// TwinCAT 3 PLC project PLCProject
// ProgramVersion: 3.1.4024.0
// libraries:
//   Tc2_MC2, * (Beckhoff Automation GmbH)
//   Tc2_NCI, * (Beckhoff Automation GmbH)
//   Tc2_NcKinematicTransformation, * (Beckhoff Automation GmbH)
//   Tc2_Standard, * (Beckhoff Automation GmbH)
//   Tc2_System, * (Beckhoff Automation GmbH)
//   Tc3_Module, * (Beckhoff Automation GmbH)
// project tree:
//   DUTs/ UI_TO_PLC.TcDUT, PLC_TO_UI.TcDUT
//   GVLs/ UIData.TcGVL
//   / PlcTask.TcTTO
//   POUs/FunctionBlock/ FB_EnableAxes.TcPOU, FB_LoadFileRun.TcPOU, FB_MachineCodeHandling.TcPOU, FB_NCIChannelGrouping.TcPOU, LifeBitMonitor.TcPOU
//   POUs/ MAIN.TcPOU
//   POUs/Programs/ Delta_Robot_Program.TcPOU
// real-time tasks:
//   TASK PlcTask: cycle T#10ms, priority 20, ADS port 350
// motion (NC):
//   TASK NC-Task 1 SAF: cycle T#2ms, priority 4, ADS port 501
//   TASK NC-Task 1 SVB: cycle T#10ms, priority 8, ADS port 511
//   AXIS X_MCS (id 1)
//   AXIS Y_MCS (id 2)
//   AXIS Z_MCS (id 3)
//   AXIS M1_ACS (id 4)
//     OtherSettings: AllowMotionCmdToSlave=true
//     encoder EncType=1
//     drive DrvType=5
//       Analog: TorqueSetpointScale=10, ScaleFactorActTorque=0.1
//     controller CtrType=1
//       CtrPara: PriorControlFactor=1
//         Observer: BandWidth=20
//   AXIS M2_ACS (id 5)
//     OtherSettings: AllowMotionCmdToSlave=true
//     encoder EncType=1
//     drive DrvType=5
//       Analog: TorqueSetpointScale=10, ScaleFactorActTorque=0.1
//     controller CtrType=1
//       CtrPara: PriorControlFactor=1
//         Observer: BandWidth=20
//   AXIS M3_ACS (id 6)
//     OtherSettings: AllowMotionCmdToSlave=true
//     encoder EncType=1
//     drive DrvType=5
//       Analog: TorqueSetpointScale=10, ScaleFactorActTorque=0.1
//     controller CtrType=1
//       CtrPara: PriorControlFactor=1
//         Observer: BandWidth=20
// variable links:
//   PLCProject Instance <-> NC-Task 1 SAF/Axes/M1_ACS
//     PlcTask Inputs/Delta_Robot_Program.io_M1.NcToPlc <-> Outputs/ToPlc
//     PlcTask Outputs/Delta_Robot_Program.io_M1.PlcToNc <-> Inputs/FromPlc
//   PLCProject Instance <-> NC-Task 1 SAF/Axes/M2_ACS
//     PlcTask Inputs/Delta_Robot_Program.io_M2.NcToPlc <-> Outputs/ToPlc
//     PlcTask Outputs/Delta_Robot_Program.io_M2.PlcToNc <-> Inputs/FromPlc
//   PLCProject Instance <-> NC-Task 1 SAF/Axes/M3_ACS
//     PlcTask Inputs/Delta_Robot_Program.io_M3.NcToPlc <-> Outputs/ToPlc
//     PlcTask Outputs/Delta_Robot_Program.io_M3.PlcToNc <-> Inputs/FromPlc
//   PLCProject Instance <-> NC-Task 1 SAF/Axes/X_MCS
//     PlcTask Inputs/Delta_Robot_Program.io_X.NcToPlc <-> Outputs/ToPlc
//     PlcTask Outputs/Delta_Robot_Program.io_X.PlcToNc <-> Inputs/FromPlc
//   PLCProject Instance <-> NC-Task 1 SAF/Axes/Y_MCS
//     PlcTask Inputs/Delta_Robot_Program.io_Y.NcToPlc <-> Outputs/ToPlc
//     PlcTask Outputs/Delta_Robot_Program.io_Y.PlcToNc <-> Inputs/FromPlc
//   PLCProject Instance <-> NC-Task 1 SAF/Axes/Z_MCS
//     PlcTask Inputs/Delta_Robot_Program.io_Z.NcToPlc <-> Outputs/ToPlc
//     PlcTask Outputs/Delta_Robot_Program.io_Z.PlcToNc <-> Inputs/FromPlc
//   PLCProject Instance <-> NC-Task 1 SAF/KinematicChannel
//     PlcTask Inputs/Delta_Robot_Program.in_stKinToPlc <-> Outputs/ToPlc
//     PlcTask Outputs/Delta_Robot_Program.out_stPlcToKin <-> Inputs/FromPlc
//   PLCProject Instance <-> NC-Task 1 SAF/NCIChannel
//     PlcTask Inputs/Delta_Robot_Program.in_stItpToPlc <-> Outputs/ToPlc
//     PlcTask Outputs/Delta_Robot_Program.out_stPlcToItp <-> Inputs/FromPlc

CONFIGURATION PLCProject
    RESOURCE PLC ON TwinCAT3
        TASK PlcTask(INTERVAL := T#10ms, PRIORITY := 20);
        PROGRAM MAIN WITH PlcTask : MAIN;
    END_RESOURCE
END_CONFIGURATION

// ---- DUTs/UI_TO_PLC.TcDUT
TYPE UI_TO_PLC :
STRUCT
	EnableMonitoring : BOOL;
	LifeBit : BOOL;
	EnableAllAxis : BOOL;
	ResetAllAxis : BOOL;
	ConfigKinematicGroup :BOOL;
	ResetKinematicGroup : BOOL;
	XJogPositive : BOOL;
	YJogPositive : BOOL;
	ZJogPositive : BOOL;
	XJogNegative : BOOL;
	YJogNegative : BOOL;
	ZJogNegative : BOOL;
	JogSpeed     : REAL;
	NCIAxisGroup : BOOL;
	NCIAxisUnGroup : BOOL;
	NCIInteperatorReset : BOOL;
	RunPartProgram : BOOL;
	StopPartProgram : BOOL;
	NCIOverRidePer : REAL;
	PartProgramName : STRING(80);
END_STRUCT
END_TYPE

// ---- DUTs/PLC_TO_UI.TcDUT
TYPE PLC_TO_UI :
STRUCT
	X_MCSPos : REAL;
	Y_MCSPos : REAL;
	Z_MCSPos : REAL;
	M1_ACSPos : REAL;
	M2_ACSPos : REAL;
	M3_ACSPos : REAL;
	AllAxisEnabled : BOOL;
	AxisError : BOOL;
	KinematicGroupError : BOOL;	
	KinematicGroupingReady : BOOL;
	NCIAxisGrouped : BOOL;
	NCIAXisError : BOOL;
	NCIInterpreterState : UDINT;
	PartProgramLine1 : STRING(80);
	PartProgramLine2 : STRING(80);
	PartProgramLine3 : STRING(80);
END_STRUCT
END_TYPE

// ---- GVLs/UIData.TcGVL
{attribute 'qualified_only'}
VAR_GLOBAL
	stUI_TO_PLC : UI_TO_PLC;
	stPLC_TO_UI : PLC_TO_UI;
END_VAR

// ---- POUs/MAIN.TcPOU
PROGRAM MAIN
VAR
END_VAR

Delta_Robot_Program();

END_PROGRAM

// ---- POUs/Programs/Delta_Robot_Program.TcPOU
PROGRAM Delta_Robot_Program
VAR	
	(* Axis Enable *)
	fbEnableAxes				: FB_EnableAxes;
	io_X						: AXIS_REF;
	io_Y						: AXIS_REF;
	io_Z						: AXIS_REF;
	io_M1						: AXIS_REF;
	io_M2						: AXIS_REF;
	io_M3						: AXIS_REF;
	bEnableAxes: BOOL;
	bAllAxesReady: BOOL;
	bAxisError: BOOL;
	bResetAxes: BOOL;
	
	(* Kinematics *)
	in_stKinToPlc	AT %I*		: NCTOPLC_NCICHANNEL_REF;
	out_stPlcToKin	AT %Q*		: PLCTONC_NCICHANNEL_REF;
	fbConfigKinGroup      		: FB_KinConfigGroup;
    stAxesConfig          		: ST_KinAxes;
	fbResetKinGroup				: FB_KinResetGroup;
	bConfigKinematicGroup: BOOL;
	bUserCartesianMode: BOOL 	:= TRUE;
	bKinGroupError: BOOL;
	bResetKinematicGroup: BOOL;
	eKinematicState: E_KINSTATUS;
	bKinematicsGroupReady: BOOL;
	
	(* Jog MCS *)
	bJogEnable: BOOL;
	fbJogAxisX					: MC_Jog;
	fbJogAxisY					: MC_Jog;
	fbJogAxisZ					: MC_Jog;
	bXJogPositive: BOOL;
	bYJogPositive: BOOL;
	bZJogPositive: BOOL;
	bXJogNegative: BOOL;
	bYJogNegative: BOOL;
	bZJogNegative: BOOL;
	rJogSpeed 	 : REAL;
	
	(* Interpolation *)
	in_stItpToPlc	AT %I*		: NCTOPLC_NCICHANNEL_REF;
	out_stPlcToItp	AT %Q*		: PLCTONC_NCICHANNEL_REF;
	fUserOverRide: LREAL := 100.0;	
	fbNCIChannelGrouping: FB_NCIChannelGrouping;
	bGroupAxes: BOOL;
	bUnGroupAxes: BOOL;
	nItpState: UDINT;
	bItpError: BOOL;
	fbIntprReset : ItpResetEx2;
	bResetInteperator: BOOL;
	bNCIAxisGrouped: BOOL;
	bNCIInteperatorError: BOOL;
	fbLoadRunStop: FB_LoadFileRun;
	bRunPRogram: BOOL;
	bStopProgram: BOOL;
	sProgramName: STRING(80):='testProgram.nc';
	bNCIProgramNotRunning: BOOL;
	
	(* UI Life Bit Monitoring *)
	fbLifeBitMonitor: LifeBitMonitor;
	lifeBitStatus: BOOL;
	exception : __SYSTEM.ExceptionCode;
	bTest: bool;
END_VAR

UI();
AxisEnable();
Kinematics();
JogMCS();
NCI();

ACTION AxisEnable:
// Enable Axes
fbEnableAxes(
	bEnableAxes					:= bEnableAxes,
	bResetAxes					:= bResetAxes, 
	io_X						:= io_X , 
	io_Y						:= io_Y , 
	io_Z						:= io_Z , 
	io_M1						:= io_M1 , 
	io_M2						:= io_M2 , 
	io_M3						:= io_M3 , 
	bAllAxesReady				=> bAllAxesReady,
	bAxisError					=> bAxisError );
END_ACTION

ACTION JogMCS:
// Manual Jogging Enable after Kinematic grouping is done & NCI program is Not Running
IF bKinematicsGroupReady AND bNCIProgramNotRunning THEN
	bJogEnable := TRUE;
ELSE
	bJogEnable := FALSE;
END_IF

fbJogAxisX(
	Axis						:= io_X, 
	JogForward					:= bXJogPositive AND bJogEnable, 
	JogBackwards				:= bXJogNegative AND bJogEnable, 
	Mode						:= MC_JOGMODE_CONTINOUS,
	Velocity					:= rJogSpeed);
	
fbJogAxisY(
	Axis						:= io_Y, 
	JogForward					:= bYJogPositive AND bJogEnable, 
	JogBackwards				:= bYJogNegative AND bJogEnable, 
	Mode						:= MC_JOGMODE_CONTINOUS,
	Velocity					:= rJogSpeed);

fbJogAxisZ(
	Axis						:= io_Z, 
	JogForward					:= bZJogPositive AND bJogEnable, 
	JogBackwards				:= bZJogNegative AND bJogEnable, 
	Mode						:= MC_JOGMODE_CONTINOUS,
	Velocity					:= rJogSpeed);
END_ACTION

ACTION Kinematics:
// Read axes id's from cylic interface
// so they can be mapped later to the kinematic group
stAxesConfig.nAxisIdsAcs[1]		:= io_M1.NcToPlc.AxisId;
stAxesConfig.nAxisIdsAcs[2]		:= io_M2.NcToPlc.AxisId;
stAxesConfig.nAxisIdsAcs[3]		:= io_M3.NcToPlc.AxisId;
stAxesConfig.nAxisIdsMcs[1]		:= io_X.NcToPlc.AxisId;
stAxesConfig.nAxisIdsMcs[2]		:= io_Y.NcToPlc.AxisId;
stAxesConfig.nAxisIdsMcs[3]		:= io_Z.NcToPlc.AxisId;

//Read Kinematics Status
eKinematicState := F_KinGetChnOperationState(stKinRefIn:=in_stKinToPlc);
IF eKinematicState = E_KINSTATUS.KinStatus_Ready THEN
	bKinematicsGroupReady := TRUE;
	bKinGroupError := FALSE;
ELSIF eKinematicState = E_KINSTATUS.KinStatus_Error THEN 
	bKinGroupError := TRUE;
	bKinematicsGroupReady := FALSE;
ELSE
	bKinematicsGroupReady := FALSE;
	bKinGroupError := FALSE	;
END_IF


// Build Kinematic Group
fbConfigKinGroup(
	bExecute					:= bConfigKinematicGroup AND bAllAxesReady AND NOT bAxisError , 
	bCartesianMode				:= bUserCartesianMode, 
	stAxesList					:= stAxesConfig, 
	stKinRefIn					:= in_stKinToPlc);

//Reset Kinematic Group
fbResetKinGroup(
	bExecute					:= bResetKinematicGroup , 
	nItpChannelId				:= in_stKinToPlc.ChnId, 
	stKinRefIn					:= in_stKinToPlc, 
	stAxesList					:= stAxesConfig);
END_ACTION

ACTION NCI:
(* Set OverRide % *)
ItpSetOverridePercent(fOverridePercent := fUserOverRide,sPlcToNci:=out_stPlcToItp);

(* Grouping Axis *)
fbNCIChannelGrouping(
	bGroupChannel:= bGroupAxes AND bKinematicsGroupReady AND bAllAxesReady AND NOT bAxisError AND NOT bItpError, 
	bUnGroupChannel:= bUnGroupAxes, 
	stX:=io_X, 
	stY:=io_Y, 
	stZ:=io_Z, 
	stItpToPlc:=in_stItpToPlc, 
	stPlcToItp:=out_stPlcToItp, 
	bBusy=> , 
	bError=> , 
	bDone=>bNCIAxisGrouped);
	
(* Inteperator State *)
nItpState := ItpGetStateInterpreter( in_stItpToPlc ); 

(* Inteperator Error *)
bNCIInteperatorError := bItpError := ItpHasError( in_stItpToPlc ); 

(* Reset Inteperator *)
fbIntprReset(
	bExecute:=bResetInteperator, 
	tTimeOut:= , 
	sNciToPlc:=in_stItpToPlc, 
	bBusy=> , 
	bErr=> , 
	nErrId=> );
	
(* Program Run & Stop NCI Program from File *)
fbLoadRunStop(
	bRun:=bRunPRogram,
	bStop :=bStopProgram,
	sPrgName:=sProgramName, 
	stItpToPlc:=in_stItpToPlc, 
	stPlcToItp:=out_stPlcToItp, 
	bBusy=> , 
	bDone=> , 
	bError=> , 
	nInterpreterState=> );
	
(* Interlock for Jog *)
IF nItpState = 1 OR nItpState = 2 THEN
	bNCIProgramNotRunning := TRUE;
ELSE
	bNCIProgramNotRunning := FALSE;
END_IF
END_ACTION

ACTION UI:
(* Life Bit Monitoring *)
IF UIData.stUI_TO_PLC.EnableMonitoring OR bTest THEN
	fbLifeBitMonitor.MonitoringTime := T#500MS;
	fbLifeBitMonitor.StartMonitor();
ELSE
	fbLifeBitMonitor.StopMonitor();
END_IF

lifeBitStatus := fbLifeBitMonitor.Status(LifeBit:=UIData.stUI_TO_PLC.LifeBit AND bTest);

IF NOT lifeBitStatus THEN
	(* For __TRY __CATCH Supported Platform *)
	(*
	__TRY
		MEMSET(destAddr:=ADR(UIData.stUI_TO_PLC.LifeBit),
		   	   fillByte:=16#0,
		   	   n:=SIZEOF(UIData.stUI_TO_PLC)-1); //SIZE - 1 is Enable Monitoring Bit size deleted
	__CATCH(exception)
			//In case of Error 
	__ENDTRY 
	*)	
	UIData.stUI_TO_PLC.EnableMonitoring := UIData.stUI_TO_PLC.LifeBit := 0;
	UIData.stUI_TO_PLC.EnableAllAxis:= UIData.stUI_TO_PLC.ResetAllAxis:= 0;
	UIData.stUI_TO_PLC.ConfigKinematicGroup:= UIData.stUI_TO_PLC.ResetKinematicGroup := 0;
	UIData.stUI_TO_PLC.XJogPositive := UIData.stUI_TO_PLC.YJogPositive := 0;
	UIData.stUI_TO_PLC.ZJogPositive := UIData.stUI_TO_PLC.XJogNegative := 0;
	UIData.stUI_TO_PLC.YJogNegative := UIData.stUI_TO_PLC.ZJogNegative:= 0;
	UIData.stUI_TO_PLC.JogSpeed := 0;
	UIData.stUI_TO_PLC.NCIAxisGroup:= 0;
	UIData.stUI_TO_PLC.NCIAxisUnGroup := UIData.stUI_TO_PLC.NCIInteperatorReset:= 0;
	UIData.stUI_TO_PLC.RunPartProgram := UIData.stUI_TO_PLC.StopPartProgram:= 0;
	UIData.stUI_TO_PLC.NCIOverRidePer := 0;
	UIData.stUI_TO_PLC.PartProgramName:= '';
	
END_IF

(*PLC to UI*)

//Position Data
UIData.stPLC_TO_UI.X_MCSPos := io_X.NcToPlc.ActPos;
UIData.stPLC_TO_UI.Y_MCSPos := io_Y.NcToPlc.ActPos;
UIData.stPLC_TO_UI.Z_MCSPos := io_Z.NcToPlc.ActPos;
UIData.stPLC_TO_UI.M1_ACSPos := io_M1.NcToPlc.ActPos;
UIData.stPLC_TO_UI.M2_ACSPos := io_M2.NcToPlc.ActPos;
UIData.stPLC_TO_UI.M3_ACSPos := io_M3.NcToPlc.ActPos;

//Axis Status
UIData.stPLC_TO_UI.AllAxisEnabled := bAllAxesReady; 
UIData.stPLC_TO_UI.AxisError := bAxisError; 
UIData.stPLC_TO_UI.KinematicGroupError := bKinGroupError;

//Kinematic Status
UIData.stPLC_TO_UI.KinematicGroupingReady := bKinematicsGroupReady;
UIData.stPLC_TO_UI.KinematicGroupError := bKinGroupError;
UIData.stPLC_TO_UI.NCIAxisGrouped := bNCIAxisGrouped;
UIData.stPLC_TO_UI.NCIAXisError := bNCIInteperatorError;
UIData.stPLC_TO_UI.NCIInterpreterState := nItpState;

(*UI to PLC*)
bEnableAxes := UIData.stUI_TO_PLC.EnableAllAxis;
bResetAxes := UIData.stUI_TO_PLC.ResetAllAxis;
bConfigKinematicGroup := UIData.stUI_TO_PLC.ConfigKinematicGroup;
bResetKinematicGroup := UIData.stUI_TO_PLC.ResetKinematicGroup;
bXJogPositive := UIData.stUI_TO_PLC.XJogPositive;
bYJogPositive := UIData.stUI_TO_PLC.YJogPositive;
bZJogPositive := UIData.stUI_TO_PLC.ZJogPositive;
bXJogNegative := UIData.stUI_TO_PLC.XJogNegative;
bYJogNegative := UIData.stUI_TO_PLC.YJogNegative;
bZJogNegative := UIData.stUI_TO_PLC.ZJogNegative;
rJogSpeed     := UIData.stUI_TO_PLC.JogSpeed;
bGroupAxes 	  := UIData.stUI_TO_PLC.NCIAxisGroup;
bUnGroupAxes  := UIData.stUI_TO_PLC.NCIAxisUnGroup;
bResetInteperator := UIData.stUI_TO_PLC.NCIInteperatorReset;
bRunPRogram 	  := UIData.stUI_TO_PLC.RunPartProgram;
bStopProgram 	  := UIData.stUI_TO_PLC.StopPartProgram;
fUserOverRide 	:= UIData.stUI_TO_PLC.NCIOverRidePer;
sProgramName := UIData.stUI_TO_PLC.PartProgramName;
END_ACTION

END_PROGRAM

// ---- POUs/FunctionBlock/FB_EnableAxes.TcPOU
FUNCTION_BLOCK FB_EnableAxes
VAR_INPUT
	bEnableAxes: BOOL;
	bResetAxes : BOOL;
END_VAR
VAR_OUTPUT
	bAllAxesReady:	BOOL:= FALSE;
	bAxisError : BOOL := FALSE;
END_VAR
VAR_IN_OUT
	io_X:	AXIS_REF;
	io_Y:	AXIS_REF;
	io_Z:	AXIS_REF;
	io_M1:	AXIS_REF;
	io_M2:	AXIS_REF;
	io_M3:	AXIS_REF;
END_VAR
VAR
	fOverride:	LREAL	:= 100.0;
	fbPowerX:	MC_Power;
	fbPowerY:	MC_Power;
	fbPowerZ:	MC_Power;
	fbPowerM1:	MC_Power;
	fbPowerM2:	MC_Power;
	fbPowerM3:	MC_Power;
	
	fbResetX:	MC_Reset;
	fbResetY:	MC_Reset;
	fbResetZ:	MC_Reset;
	fbResetM1:	MC_Reset;
	fbResetM2:	MC_Reset;
	fbResetM3:	MC_Reset;
	
	
	m: MC_Reset;
END_VAR

io_X.ReadStatus();
io_Y.ReadStatus();
io_Z.ReadStatus();
io_M1.ReadStatus();
io_M2.ReadStatus();
io_M3.ReadStatus();


fbPowerX(
	Enable				:= bEnableAxes, 
	Enable_Positive		:= bEnableAxes, 
	Enable_Negative		:= bEnableAxes, 
	Override			:= fOverride,
	BufferMode			:= MC_Aborting,
	Axis				:= io_X);

fbPowerY(
	Enable				:= bEnableAxes, 
	Enable_Positive		:= bEnableAxes, 
	Enable_Negative		:= bEnableAxes, 
	Override			:= fOverride,
	BufferMode			:= MC_Aborting,
	Axis				:= io_Y);
	
fbPowerZ(
	Enable				:= bEnableAxes, 
	Enable_Positive		:= bEnableAxes, 
	Enable_Negative		:= bEnableAxes, 
	Override			:= fOverride,
	BufferMode			:= MC_Aborting,
	Axis				:= io_Z);
	
fbPowerM1(
	Enable				:= bEnableAxes, 
	Enable_Positive		:= bEnableAxes, 
	Enable_Negative		:= bEnableAxes, 
	Override			:= fOverride,
	BufferMode			:= MC_Aborting,
	Axis				:= io_M1);
	
fbPowerM2(
	Enable				:= bEnableAxes, 
	Enable_Positive		:= bEnableAxes, 
	Enable_Negative		:= bEnableAxes, 
	Override			:= fOverride,
	BufferMode			:= MC_Aborting,
	Axis				:= io_M2);
	
fbPowerM3(
	Enable				:= bEnableAxes, 
	Enable_Positive		:= bEnableAxes, 
	Enable_Negative		:= bEnableAxes, 
	Override			:= fOverride,
	BufferMode			:= MC_Aborting,
	Axis				:= io_M3);
	
fbResetX(
	Axis:=io_X, 
	Execute:=bResetAxes, 
	Done=> , 
	Busy=> , 
	Error=> , 
	ErrorID=> );
	
fbResetY(
	Axis:=io_Y, 
	Execute:=bResetAxes, 
	Done=> , 
	Busy=> , 
	Error=> , 
	ErrorID=> );
	
fbResetZ(
	Axis:=io_Z, 
	Execute:=bResetAxes, 
	Done=> , 
	Busy=> , 
	Error=> , 
	ErrorID=> );
	
fbResetM1(
	Axis:=io_M1, 
	Execute:=bResetAxes, 
	Done=> , 
	Busy=> , 
	Error=> , 
	ErrorID=> );
	
fbResetM2(
	Axis:=io_M2, 
	Execute:=bResetAxes, 
	Done=> , 
	Busy=> , 
	Error=> , 
	ErrorID=> );
	
fbResetM3(
	Axis:=io_M3, 
	Execute:=bResetAxes, 
	Done=> , 
	Busy=> , 
	Error=> , 
	ErrorID=> );
	
bAllAxesReady	:=	fbPowerX.Status AND fbPowerY.Status AND fbPowerZ.Status
					AND	fbPowerM1.Status AND fbPowerM2.Status AND fbPowerM3.Status;
					
bAxisError      := fbPowerX.Error OR fbPowerY.Error OR fbPowerZ.Error 
				   OR fbPowerM1.Error OR fbPowerM2.Error OR fbPowerM3.Error;

END_FUNCTION_BLOCK

// ---- POUs/FunctionBlock/FB_NCIChannelGrouping.TcPOU
FUNCTION_BLOCK FB_NCIChannelGrouping
VAR_INPUT
	bGroupChannel : BOOL;
	bUnGroupChannel: BOOL;
END_VAR
VAR_IN_OUT
	stX	: AXIS_REF;
	stY	: AXIS_REF;
	stZ	: AXIS_REF;
	stItpToPlc : NCTOPLC_NCICHANNEL_REF;
	stPlcToItp : PLCTONC_NCICHANNEL_REF;
END_VAR
VAR_OUTPUT
	bBusy : BOOL;
	bError : BOOL;
	bDone : BOOL;
	
END_VAR
VAR
	nState: INT;
	nErrorState: INT;
	fbBuildNCIGroup: CfgBuild3DGroup;

	fbDeGroupNCI: CfgReconfigGroup;
END_VAR

CASE nState OF
	0:
		IF bGroupChannel AND NOT bDone THEN
			bBusy := FALSE;
			bError := FALSE;
			bDone := FALSE;
			nErrorState := nState;
			nState := 10;
		END_IF
		IF bUnGroupChannel THEN
			bBusy := FALSE;
			bError := FALSE;
			bDone := FALSE;
			nErrorState := nState;
			nState := 110;
		END_IF
	
	10:
	
		fbBuildNCIGroup(
			bExecute:= TRUE, 
			nGroupId:= ItpGetGroupId(sNciToPlc:=stItpToPlc), 
			nXAxisId:=stX.NcToPlc.AxisId, 
			nYAxisId:=stY.NcToPlc.AxisId, 
			nZAxisId:=stZ.NcToPlc.AxisId,
			tTimeOut:= , 
			bBusy=> , 
			bErr=> , 
			nErrId=> );
		IF NOT fbBuildNCIGroup.bBusy THEN
			IF NOT fbBuildNCIGroup.bErr THEN
				nState	:= 20;
			ELSE
				(* add error handling *)
				nErrorState	:= nState;
				bBusy	:= FALSE;
				bError	:= TRUE;
				nState	:= 9000;
			END_IF
			fbBuildNCIGroup(bExecute:=FALSE); 
		END_IF
	20:
		bDone := TRUE;
		nState	:= 9000;
	
	110:
	
		fbDeGroupNCI(
			bExecute:= TRUE , 
			nGroupId:=ItpGetGroupId(sNciToPlc:=stItpToPlc), 
			tTimeOut:= , 
			bBusy=> , 
			bErr=> , 
			nErrId=> );
		IF NOT fbDeGroupNCI.bBusy THEN
			IF NOT fbDeGroupNCI.bErr THEN
				nState := 120;
			ELSE
				(* ADD error handling *)
				nErrorState	:= nState;
				bBusy	:= FALSE;
				bError	:= TRUE;
				nState	:= 9500;
			END_IF
			fbDeGroupNCI(bExecute:=FALSE);
		END_IF
		
	120:
		bDone := FALSE;
		nState	:= 9500;	
	
	9000:
	// error state 
	IF NOT bGroupChannel THEN
		nState	:= 0;
		bError	:= FALSE;
	END_IF
	
	9500:
	// error state 
	IF NOT bUnGroupChannel THEN
		nState	:= 0;
		bError	:= FALSE;
	END_IF
	
	
END_CASE

END_FUNCTION_BLOCK

// ---- POUs/FunctionBlock/FB_LoadFileRun.TcPOU
FUNCTION_BLOCK FB_LoadFileRun
VAR_INPUT
	bRun: BOOL;
	sPrgName : STRING(255);
	bStop : BOOL;
END_VAR
VAR_IN_OUT
	stItpToPlc			: NCTOPLC_NCICHANNEL_REF;
	stPlcToItp			: PLCTONC_NCICHANNEL_REF;
END_VAR
VAR_OUTPUT
	bBusy: BOOL;
	bDone: BOOL;
	bError: BOOL;
	nInterpreterState	: UDINT	:= 0;
END_VAR
VAR
	fbLoadGCode			: ItpLoadProgEx;
	fbStartGCode		: ItpStartStopEx;
	nState: INT;
	nErrorState: INT;
	stopRisingEdge : R_TRIG;
END_VAR

stopRisingEdge(CLK:=bStop);
IF stopRisingEdge.Q THEN
	bBusy:= TRUE;
	bDone:= FALSE;
	nState := 80;
END_IF

CASE nState OF
	0:
		IF bRun AND NOT bStop THEN
			bBusy	:= TRUE;
			bDone	:= FALSE;
			bError	:= FALSE;
			nErrorState	:= nState;
			nState	:= 20;
		END_IF
	
	20:
	// load g-code file 
	// pls. ensure that first.nc is available in TwinCAT\MC\NCI-folder 
	fbLoadGCode(
		sNciToPlc:=stItpToPlc, 
		bExecute:=TRUE, 
		sPrg:= sPrgName, 
		nLength:= INT_TO_UDINT(LEN(sPrgName)), 
		tTimeOut:= , 
		bBusy=> , 
		bErr=> , 
		nErrId=> );
	IF NOT fbLoadGCode.bBusy THEN
		IF NOT fbLoadGCode.bErr THEN
			nState	:= 30;
		ELSE
			(* add error handling *)
			nErrorState	:= nState;
			bBusy	:= FALSE;
			bError	:= TRUE;
			nState	:= 9999;				
		END_IF
		fbLoadGCode(sNciToPlc:=stItpToPlc, bExecute:=FALSE); 
	END_IF
	
	30:
		// we have to check the status of the interpreter. It has to be in ready state, in case of loading the program successfully.
		nInterpreterState	:= ItpGetStateInterpreter(sNciToPlc:=stItpToPlc);
		IF nInterpreterState = Tc2_NCI.NCI_INTERPRETER_READY THEN
			nState	:= 40;
		ELSE
			(* add error handling *)
			nErrorState	:= nState;
			bBusy	:= FALSE;
			bError	:= TRUE;
			nState	:= 9999;				
		END_IF
		
	40:
		// start g-code file
		fbStartGCode(
			bStart:=TRUE, 
			bStop:=FALSE, 
			tTimeOut:= , 
			sNciToPlc:= stItpToPlc, 
			bBusy=> , 
			bErr=> , 
			nErrId=> );
		IF NOT fbStartGCode.bBusy THEN
			IF NOT fbStartGCode.bErr THEN
				nState	:= 50;
			ELSE	
				(* add error handling *)
				nErrorState	:= nState;
				bBusy	:= FALSE;
				bError	:= TRUE;
				nState	:= 9999;				
			END_IF
			fbStartGCode( bStart:=FALSE, sNciToPlc:= stItpToPlc ); 
		END_IF
		
	50:
		// check state, again - we are at least not in ready state for several ticks
		// this is to ensure that we don't indicate program has finished, before we have started 
		nInterpreterState	:= ItpGetStateInterpreter(sNciToPlc:=stItpToPlc);
		IF nInterpreterState <> Tc2_NCI.NCI_INTERPRETER_READY THEN
			// nci is running
			nState	:= 60;
		END_IF
	
	60:
		nInterpreterState	:= ItpGetStateInterpreter(sNciToPlc:=stItpToPlc);
		IF	nInterpreterState = Tc2_NCI.NCI_INTERPRETER_READY THEN
			// program has finished
			nState	:= 70;
		ELSIF nInterpreterState = Tc2_NCI.NCI_INTERPRETER_ABORTED THEN
			// a run-time error occured - this could be a lag error or something else... 
			// add error handling
			;
		END_IF	
	70:
		bDone	:= TRUE;
		bBusy	:= FALSE;
		IF NOT bRun THEN
			nState	:= 0;
		END_IF
	80:
		fbLoadGCode(
			sNciToPlc:=stItpToPlc, 
			bExecute:=FALSE);
		fbStartGCode(
			bStart:=FALSE, 
			bStop:=FALSE, 
			tTimeOut:= , 
			sNciToPlc:= stItpToPlc);
		IF NOT fbLoadGCode.bBusy AND NOT fbStartGCode.bBusy THEN
			nState := 90;
		ELSE
			nState := 9999;
		END_IF
	90:
		// Stop g-code file
		fbStartGCode(
			bStart:=FALSE, 
			bStop:=TRUE, 
			tTimeOut:= , 
			sNciToPlc:= stItpToPlc, 
			bBusy=> , 
			bErr=> , 
			nErrId=> );
		IF NOT fbStartGCode.bBusy THEN
			IF NOT fbStartGCode.bErr THEN
				nState	:= 0;
			ELSE	
				(* add error handling *)
				nErrorState	:= nState;
				bBusy	:= FALSE;
				bError	:= TRUE;
				nState	:= 9999;				
			END_IF
			fbStartGCode( bStop:=FALSE, sNciToPlc:= stItpToPlc );
			bBusy := FALSE; 
		END_IF
	9999:
		// error state 
		IF NOT bRun THEN
			nState	:= 0;
			bError	:= FALSE;
		END_IF
END_CASE

END_FUNCTION_BLOCK

// ---- POUs/FunctionBlock/LifeBitMonitor.TcPOU
FUNCTION_BLOCK LifeBitMonitor
VAR
	_EnableMonitoring : BOOL;
	_MonitoringTime : TIME;
	_LifeBitLostCount  : INT;
END_VAR

PROPERTY MonitoringTime : TIME
SET
_MonitoringTime := MonitoringTime;
END_SET
END_PROPERTY

METHOD StartMonitor : BOOL
_EnableMonitoring := TRUE;
END_METHOD

METHOD Status : BOOL
VAR_INPUT
	LifeBit : BOOL;
END_VAR
VAR_INST
    LifeBitTimer  : TON;
	LifeBitLast : BOOL;
END_VAR
IF _EnableMonitoring THEN
	(* Reset Timer on LifeBit Toggle *)
	IF LifeBit AND NOT LifeBitLast THEN
		 LifeBitTimer(IN := FALSE);
	END_IF
	
	(* Store the last state of LifeBit *)
	LifeBitLast := LifeBit;
	
	(* Start the Timer *)
	LifeBitTimer(IN := TRUE, PT := _MonitoringTime);
	
	(* Update Communication Status *)
	IF LifeBitTimer.Q THEN
		Status := FALSE;            (* Communication failed *)
	ELSE
		Status := TRUE;             (* Communication is OK *)
	END_IF;
ELSE
    LifeBitTimer(IN := FALSE);      (* Ensure timer is off when monitoring is off *)
	Status := FALSE;
END_IF
END_METHOD

METHOD StopMonitor : BOOL
_EnableMonitoring := FALSE;
END_METHOD

END_FUNCTION_BLOCK

// ---- POUs/FunctionBlock/FB_MachineCodeHandling.TcPOU
FUNCTION_BLOCK FB_MachineCodeHandling
VAR_INPUT
	
END_VAR
VAR_OUTPUT
END_VAR
VAR_IN_OUT
	 sNciToPlc      : NCTOPLC_NCICHANNEL_REF;
	 sPlcToNci      : PLCTONC_NCICHANNEL_REF;
END_VAR
VAR
	 bMFuncRequest: BOOL;
	 nMCode: INT;
	 bM100Requested: BOOL;
	 bM100Done: BOOL;
	 MCodeConfirm: ItpConfirmHsk;
	 bModeConfirm: BOOL;
	 bMCodeConfirmError: BOOL;
	 nErrorID: UDINT;
	 bResetMCodeConfirm: BOOL;
	 nToolNumber: UINT;
END_VAR

(*
Sample NC Program
G00 X5 Y5                
G01 X0 Y20 F200  
M100 T5        M100 is Tool Change Code & T5 is the Tool Number
G01 X20 Y0               
M30          
*)

(* Check M-Code Present *)
bMFuncRequest := ItpIsHskMFunc(sNciToPlc ); 

(* Get M-Code Number *)
IF bMFuncRequest THEN
	nMCode := ItpGetHskMFunc(sNciToPlc);
ELSE
	nMCode := 0;
END_IF

(* Get Tool Number *)
nToolNumber := ItpGetTParam(sNciToPlc);

(* MCode M100 *)
IF bMFuncRequest AND nMCode = 100 THEN
	bM100Requested := TRUE; 
END_IF
//User Defined M Code Program
IF bM100Requested THEN
	//Your logic
END_IF
//User Defined M Code Confirm
IF  bM100Done THEN
	bM100Requested := FALSE; 
	bModeConfirm := TRUE;
	bM100Done := FALSE;
END_IF

//Confirm M-Code Common for all M-Code
MCodeConfirm(
		bExecute:=bModeConfirm AND NOT bMCodeConfirmError , 
		sNciToPlc:=sNciToPlc, 
		sPlcToNci:=sPlcToNci, 
		bBusy=> , 
		bErr=> , 
		nErrId=> );

IF bModeConfirm THEN
	IF NOT MCodeConfirm.bBusy THEN
		IF MCodeConfirm.bErr THEN
			bMCodeConfirmError := TRUE;
			nErrorID := MCodeConfirm.nErrId ;
		ELSE
			bModeConfirm := FALSE;
		END_IF
	END_IF
END_IF

IF bResetMCodeConfirm THEN
	bResetMCodeConfirm := FALSE;
	bMCodeConfirmError := FALSE;
	nErrorID := 0 ;
END_IF

END_FUNCTION_BLOCK
